FUNCTION UpdateEventTimeStampWithSystemTime
VAR_INPUT
	stEvent: REFERENCE TO ST_Event;
 
END_VAR
VAR
	//timeStruct: TIMESTRUCT;
	 //LocalSystemTime: FB_LocalSystemTime();
	 fbGetsytstemtime: GETSYSTEMTIME;
	 filetime: T_FILETIME;
END_VAR


//LocalSystemTime(bEnable:=TRUE,systemTime=> timeStruct);
//timeStruct;
fbGetsytstemtime(timeLoDW=> filetime.dwLowDateTime, timeHiDW=> filetime.dwHighDateTime);//SYSTEMTIME_TO_DT(TIMESTR:=timeStruct);
stEvent.dtTimeStamp:= FILETIME_TO_DT(filetime);

END_FUNCTION

(* stored: Version 1.1.0.1, ProductVersion 3.1.4024.11
   POU UpdateEventTimeStampWithSystemTime: Id {628cd157-4255-40a9-9c5d-2aa26c45db05}, SpecialFunc None *)
